// TwinCAT 3 PLC project Linearachse
// ProgramVersion: 3.1.4022.1
// libraries:
//   Tc2_Standard, * (Beckhoff Automation GmbH)
//   Tc2_System, * (Beckhoff Automation GmbH)
//   Tc3_Module, * (Beckhoff Automation GmbH)
// project tree:
//   GVLs/ Sim.TcGVL
//   / PlcTask.TcTTO (not stored)
//   POUs/ Linearachse.TcPOU, MAIN.TcPOU
//   Privat/ DatenRangieren.TcPOU, Hardware.TcGVL, Computer.TcGVL
// real-time tasks:
//   TASK PlcTask: cycle T#10ms, priority 20, ADS port 350
// motion (NC):
//   TASK NC-Task 1 SAF: cycle T#2ms, priority 4, ADS port 501
//   TASK NC-Task 1 SVB: cycle T#10ms, priority 8, ADS port 511
//   AXIS Axis 1 (id 1)
//     OtherSettings: AllowMotionCmdToSlave=true
//     encoder EncType=4
//       EncPara: MaxCount=#x0000ffff
//         Inc: RefSoftSyncMask=#x0000ffff
//     drive DrvType=24
//       Analog: ScaleFactorActTorque=0.1
//       TimeComp: TaskDelayCycles=1
//     controller CtrType=1
//       CtrPara: PriorControlFactor=1
//         Observer: BandWidth=20
//   AXIS Axis 2 (id 2)
//     OtherSettings: AllowMotionCmdToSlave=true
//     encoder EncType=4
//       EncPara: MaxCount=#x0000ffff
//         Inc: RefSoftSyncMask=#x0000ffff
//     drive DrvType=24
//       Analog: ScaleFactorActTorque=0.1
//       TimeComp: TaskDelayCycles=1
//     controller CtrType=1
//       CtrPara: PriorControlFactor=1
//         Observer: BandWidth=20
//   AXIS Axis 3 (id 3)
//     OtherSettings: AllowMotionCmdToSlave=true
//     encoder EncType=4
//       EncPara: MaxCount=#x0000ffff
//     drive DrvType=23
//       Analog: ScaleFactorActTorque=0.1
//       TimeComp: TaskDelayCycles=1
//     controller CtrType=1
//       CtrPara: PriorControlFactor=1
//         Observer: BandWidth=20
//   AXIS Axis 4 (id 4)
//     OtherSettings: AllowMotionCmdToSlave=true
//     encoder EncType=4
//       EncPara: MaxCount=#x0000ffff
//     drive DrvType=23
//       Analog: ScaleFactorActTorque=0.1
//       TimeComp: TaskDelayCycles=1
//     controller CtrType=1
//       CtrPara: PriorControlFactor=1
//         Observer: BandWidth=20
//   AXIS Axis 5 (id 5)
//     OtherSettings: AllowMotionCmdToSlave=true
//     encoder EncType=19
//       EncPara: MaxCount=#xffffffff
//     drive DrvType=16
//       DrvPara: MaxCount=#xffffffff
//         Analog: ScaleFactorActTorque=0.1
//         TimeComp: TaskDelayCycles=1
//     controller CtrType=1
//       CtrPara: PriorControlFactor=1
//         Observer: BandWidth=20
//   AXIS Axis 6 (id 6)
//     OtherSettings: AllowMotionCmdToSlave=true
//     encoder EncType=19
//       EncPara: MaxCount=#xffffffff
//     drive DrvType=16
//       DrvPara: MaxCount=#xffffffff
//         Analog: ScaleFactorActTorque=0.1
//         TimeComp: TaskDelayCycles=1
//     controller CtrType=1
//       CtrPara: PriorControlFactor=1
//         Observer: BandWidth=20
// I/O:
//   DEVICE Device 1 (EtherCAT), AmsNetId 192.168.0.200.2.1
//     Term 1 (EK1200) [EK1200-5000 EtherCAT Power supply (2A E-Bus)]
//       Term 2 (EL1809) [EL1809 16Ch. Dig. Input 24V, 3ms]
//       Term 3 (EL1809) [EL1809 16Ch. Dig. Input 24V, 3ms]
//       Term 4 (EL2809) [EL2809 16Ch. Dig. Output 24V, 0.5A]
//       Term 5 (EL2809) [EL2809 16Ch. Dig. Output 24V, 0.5A]
//       Term 6 (EL3064) [EL3064 4Ch. Ana. Input 0-10V]
//       Term 7 (EL4034) [EL4034 4Ch. Ana. Output +/-10V, 12bit]
//       Term 8 (EL7031) [EL7031 1Ch. Stepper motor output stage (24V, 1.5A)]
//       Term 9 (EL7031) [EL7031 1Ch. Stepper motor output stage (24V, 1.5A)]
//       Term 10 (EL7332) [EL7332 2Ch. DC motor output stage (24V, 1.5A)]
//       Term 11 (EL7201-0010) [EL7201-0010 1Ch. MDP742 Servo motor output stage with OCT (50V, 4A)]
//       Term 12 (EL7201-0010) [EL7201-0010 1Ch. MDP742 Servo motor output stage with OCT (50V, 4A)]
//       Term 26 (EL6090) [EL6090 Display terminal]
//       Term 27 (EK1110) [EK1110 EtherCAT extension]
// variable links:
//   NC-Task 1 SAF/Axes/Axis 1 <-> Device 1 (EtherCAT)/Term 1 (EK1200)/Term 8 (EL7031)
//     Drive/Inputs/In/nState1 @bit 3 <-> STM Status/Status/Error
//     Drive/Inputs/In/nState1 @bit 5 <-> STM Status/Status/Moving negative
//     Drive/Inputs/In/nState1 @bit 4 <-> STM Status/Status/Moving positive
//     Drive/Inputs/In/nState1 @bit 1 <-> STM Status/Status/Ready
//     Drive/Inputs/In/nState1 <-> STM Status/Status/Ready to enable
//     Drive/Inputs/In/nState1 @bit 6 <-> STM Status/Status/Torque reduced
//     Drive/Inputs/In/nState1 @bit 2 <-> STM Status/Status/Warning
//     Drive/Inputs/In/nState2 @bit 3 <-> STM Status/Status/Digital input 1
//     Drive/Inputs/In/nState2 @bit 4 <-> STM Status/Status/Digital input 2
//     Drive/Inputs/In/nState2 @bit 5 <-> STM Status/Status/Sync error
//     Drive/Inputs/In/nState2 @bit 7 <-> STM Status/Status/TxPDO Toggle
//     Drive/Inputs/In/nState4 @bit 1 <-> WcState/InputToggle
//     Drive/Inputs/In/nState4 <-> WcState/WcState
//     Drive/Outputs/Out/nCtrl1 <-> STM Control/Control/Enable
//     Drive/Outputs/Out/nCtrl1 @bit 2 <-> STM Control/Control/Reduce torque
//     Drive/Outputs/Out/nCtrl1 @bit 1 <-> STM Control/Control/Reset
//     Drive/Outputs/Out/nDataOut2[0] <-> STM Velocity/Velocity
//     Enc/Inputs/In/nDataIn1[0] <-> ENC Status compact/Counter value
//     Enc/Inputs/In/nDataIn2[0] <-> ENC Status compact/Latch value
//     Enc/Inputs/In/nState1 @bit 4 <-> ENC Status compact/Status/Counter overflow
//     Enc/Inputs/In/nState1 @bit 3 <-> ENC Status compact/Status/Counter underflow
//     Enc/Inputs/In/nState1 @bit 1 <-> ENC Status compact/Status/Latch extern valid
//     Enc/Inputs/In/nState1 @bit 2 <-> ENC Status compact/Status/Set counter done
//     Enc/Inputs/In/nState2 @bit 4 <-> ENC Status compact/Status/Status of extern latch
//     Enc/Inputs/In/nState2 @bit 5 <-> ENC Status compact/Status/Sync error
//     Enc/Inputs/In/nState2 @bit 7 <-> ENC Status compact/Status/TxPDO Toggle
//     Enc/Inputs/In/nState4 @bit 1 <-> WcState/InputToggle
//     Enc/Inputs/In/nState4 <-> WcState/WcState
//     Enc/Outputs/Out/nCtrl1 @bit 3 <-> ENC Control compact/Control/Enable latch extern on negative edge
//     Enc/Outputs/Out/nCtrl1 @bit 1 <-> ENC Control compact/Control/Enable latch extern on positive edge
//     Enc/Outputs/Out/nCtrl1 @bit 2 <-> ENC Control compact/Control/Set counter
//     Enc/Outputs/Out/nDataOut1[0] <-> ENC Control compact/Set counter value
//   NC-Task 1 SAF/Axes/Axis 2 <-> Device 1 (EtherCAT)/Term 1 (EK1200)/Term 9 (EL7031)
//     Drive/Inputs/In/nState1 @bit 3 <-> STM Status/Status/Error
//     Drive/Inputs/In/nState1 @bit 5 <-> STM Status/Status/Moving negative
//     Drive/Inputs/In/nState1 @bit 4 <-> STM Status/Status/Moving positive
//     Drive/Inputs/In/nState1 @bit 1 <-> STM Status/Status/Ready
//     Drive/Inputs/In/nState1 <-> STM Status/Status/Ready to enable
//     Drive/Inputs/In/nState1 @bit 6 <-> STM Status/Status/Torque reduced
//     Drive/Inputs/In/nState1 @bit 2 <-> STM Status/Status/Warning
//     Drive/Inputs/In/nState2 @bit 3 <-> STM Status/Status/Digital input 1
//     Drive/Inputs/In/nState2 @bit 4 <-> STM Status/Status/Digital input 2
//     Drive/Inputs/In/nState2 @bit 5 <-> STM Status/Status/Sync error
//     Drive/Inputs/In/nState2 @bit 7 <-> STM Status/Status/TxPDO Toggle
//     Drive/Inputs/In/nState4 @bit 1 <-> WcState/InputToggle
//     Drive/Inputs/In/nState4 <-> WcState/WcState
//     Drive/Outputs/Out/nCtrl1 <-> STM Control/Control/Enable
//     Drive/Outputs/Out/nCtrl1 @bit 2 <-> STM Control/Control/Reduce torque
//     Drive/Outputs/Out/nCtrl1 @bit 1 <-> STM Control/Control/Reset
//     Drive/Outputs/Out/nDataOut2[0] <-> STM Velocity/Velocity
//     Enc/Inputs/In/nDataIn1[0] <-> ENC Status compact/Counter value
//     Enc/Inputs/In/nDataIn2[0] <-> ENC Status compact/Latch value
//     Enc/Inputs/In/nState1 @bit 4 <-> ENC Status compact/Status/Counter overflow
//     Enc/Inputs/In/nState1 @bit 3 <-> ENC Status compact/Status/Counter underflow
//     Enc/Inputs/In/nState1 @bit 1 <-> ENC Status compact/Status/Latch extern valid
//     Enc/Inputs/In/nState1 @bit 2 <-> ENC Status compact/Status/Set counter done
//     Enc/Inputs/In/nState2 @bit 4 <-> ENC Status compact/Status/Status of extern latch
//     Enc/Inputs/In/nState2 @bit 5 <-> ENC Status compact/Status/Sync error
//     Enc/Inputs/In/nState2 @bit 7 <-> ENC Status compact/Status/TxPDO Toggle
//     Enc/Inputs/In/nState4 @bit 1 <-> WcState/InputToggle
//     Enc/Inputs/In/nState4 <-> WcState/WcState
//     Enc/Outputs/Out/nCtrl1 @bit 3 <-> ENC Control compact/Control/Enable latch extern on negative edge
//     Enc/Outputs/Out/nCtrl1 @bit 1 <-> ENC Control compact/Control/Enable latch extern on positive edge
//     Enc/Outputs/Out/nCtrl1 @bit 2 <-> ENC Control compact/Control/Set counter
//     Enc/Outputs/Out/nDataOut1[0] <-> ENC Control compact/Set counter value
//   NC-Task 1 SAF/Axes/Axis 3 <-> Device 1 (EtherCAT)/Term 1 (EK1200)/Term 10 (EL7332)
//     Drive/Inputs/In/nState1 @bit 3 <-> DCM Status Channel 1/Status/Error
//     Drive/Inputs/In/nState1 @bit 5 <-> DCM Status Channel 1/Status/Moving negative
//     Drive/Inputs/In/nState1 @bit 4 <-> DCM Status Channel 1/Status/Moving positive
//     Drive/Inputs/In/nState1 @bit 1 <-> DCM Status Channel 1/Status/Ready
//     Drive/Inputs/In/nState1 <-> DCM Status Channel 1/Status/Ready to enable
//     Drive/Inputs/In/nState1 @bit 6 <-> DCM Status Channel 1/Status/Torque reduced
//     Drive/Inputs/In/nState1 @bit 2 <-> DCM Status Channel 1/Status/Warning
//     Drive/Inputs/In/nState2 @bit 3 <-> DCM Status Channel 1/Status/Digital input 1
//     Drive/Inputs/In/nState2 @bit 4 <-> DCM Status Channel 1/Status/Digital input 2
//     Drive/Inputs/In/nState2 @bit 5 <-> DCM Status Channel 1/Status/Sync error
//     Drive/Inputs/In/nState2 @bit 7 <-> DCM Status Channel 1/Status/TxPDO Toggle
//     Drive/Inputs/In/nState4 @bit 1 <-> WcState/InputToggle
//     Drive/Inputs/In/nState4 <-> WcState/WcState
//     Drive/Outputs/Out/nCtrl1 <-> DCM Control Channel 1/Control/Enable
//     Drive/Outputs/Out/nCtrl1 @bit 2 <-> DCM Control Channel 1/Control/Reduce torque
//     Drive/Outputs/Out/nCtrl1 @bit 1 <-> DCM Control Channel 1/Control/Reset
//     Drive/Outputs/Out/nDataOut2[0] <-> DCM Velocity Channel 1/Velocity
//   NC-Task 1 SAF/Axes/Axis 4 <-> Device 1 (EtherCAT)/Term 1 (EK1200)/Term 10 (EL7332)
//     Drive/Inputs/In/nState1 @bit 3 <-> DCM Status Channel 2/Status/Error
//     Drive/Inputs/In/nState1 @bit 5 <-> DCM Status Channel 2/Status/Moving negative
//     Drive/Inputs/In/nState1 @bit 4 <-> DCM Status Channel 2/Status/Moving positive
//     Drive/Inputs/In/nState1 @bit 1 <-> DCM Status Channel 2/Status/Ready
//     Drive/Inputs/In/nState1 <-> DCM Status Channel 2/Status/Ready to enable
//     Drive/Inputs/In/nState1 @bit 6 <-> DCM Status Channel 2/Status/Torque reduced
//     Drive/Inputs/In/nState1 @bit 2 <-> DCM Status Channel 2/Status/Warning
//     Drive/Inputs/In/nState2 @bit 3 <-> DCM Status Channel 2/Status/Digital input 1
//     Drive/Inputs/In/nState2 @bit 4 <-> DCM Status Channel 2/Status/Digital input 2
//     Drive/Inputs/In/nState2 @bit 5 <-> DCM Status Channel 2/Status/Sync error
//     Drive/Inputs/In/nState2 @bit 7 <-> DCM Status Channel 2/Status/TxPDO Toggle
//     Drive/Inputs/In/nState4 @bit 1 <-> WcState/InputToggle
//     Drive/Inputs/In/nState4 <-> WcState/WcState
//     Drive/Outputs/Out/nCtrl1 <-> DCM Control Channel 2/Control/Enable
//     Drive/Outputs/Out/nCtrl1 @bit 2 <-> DCM Control Channel 2/Control/Reduce torque
//     Drive/Outputs/Out/nCtrl1 @bit 1 <-> DCM Control Channel 2/Control/Reset
//     Drive/Outputs/Out/nDataOut2[0] <-> DCM Velocity Channel 2/Velocity
//   NC-Task 1 SAF/Axes/Axis 5 <-> Device 1 (EtherCAT)/Term 1 (EK1200)/Term 11 (EL7201-0010)
//     Drive/Inputs/In/nDcOutputTime <-> InfoData/DcOutputShift
//     Drive/Inputs/In/nState1 <-> DRV Statusword/Statusword
//     Drive/Inputs/In/nState2 <-> DRV Statusword/Statusword @bit 8
//     Drive/Inputs/In/nState4 @bit 1 <-> WcState/InputToggle
//     Drive/Inputs/In/nState4 <-> WcState/WcState
//     Drive/Outputs/Out/nCtrl1 <-> DRV Controlword/Controlword
//     Drive/Outputs/Out/nCtrl2 <-> DRV Controlword/Controlword @bit 8
//     Drive/Outputs/Out/nDataOut2 <-> DRV Target velocity/Target velocity
//     Enc/Inputs/In/nDataIn1 <-> FB Position/Position
//     Enc/Inputs/In/nDcInputTime <-> InfoData/DcInputShift
//     Enc/Inputs/In/nState4 @bit 1 <-> WcState/InputToggle
//     Enc/Inputs/In/nState4 <-> WcState/WcState
//   NC-Task 1 SAF/Axes/Axis 6 <-> Device 1 (EtherCAT)/Term 1 (EK1200)/Term 12 (EL7201-0010)
//     Drive/Inputs/In/nDcOutputTime <-> InfoData/DcOutputShift
//     Drive/Inputs/In/nState1 <-> DRV Statusword/Statusword
//     Drive/Inputs/In/nState2 <-> DRV Statusword/Statusword @bit 8
//     Drive/Inputs/In/nState4 @bit 1 <-> WcState/InputToggle
//     Drive/Inputs/In/nState4 <-> WcState/WcState
//     Drive/Outputs/Out/nCtrl1 <-> DRV Controlword/Controlword
//     Drive/Outputs/Out/nCtrl2 <-> DRV Controlword/Controlword @bit 8
//     Drive/Outputs/Out/nDataOut2 <-> DRV Target velocity/Target velocity
//     Enc/Inputs/In/nDataIn1 <-> FB Position/Position
//     Enc/Inputs/In/nDcInputTime <-> InfoData/DcInputShift
//     Enc/Inputs/In/nState4 @bit 1 <-> WcState/InputToggle
//     Enc/Inputs/In/nState4 <-> WcState/WcState
//   Linearachse/Linearachse Instance <-> Device 1 (EtherCAT)/Term 1 (EK1200)/Term 2 (EL1809)
//     PlcTask Inputs/Hardware.DI_0_1_bis_8 <-> Channel 1/Input
//     PlcTask Inputs/Hardware.DI_0_9_bis_16 <-> Channel 8/Input
//     PlcTask Inputs/Hardware.DI_0_1_bis_8 @bit 1 <-> Channel 2/Input
//     PlcTask Inputs/Hardware.DI_0_1_bis_8 @bit 2 <-> Channel 3/Input
//     PlcTask Inputs/Hardware.DI_0_1_bis_8 @bit 3 <-> Channel 4/Input
//     PlcTask Inputs/Hardware.DI_0_1_bis_8 @bit 4 <-> Channel 5/Input
//     PlcTask Inputs/Hardware.DI_0_1_bis_8 @bit 5 <-> Channel 6/Input
//     PlcTask Inputs/Hardware.DI_0_1_bis_8 @bit 6 <-> Channel 7/Input
//     PlcTask Inputs/Hardware.DI_0_9_bis_16 @bit 1 <-> Channel 10/Input
//     PlcTask Inputs/Hardware.DI_0_9_bis_16 @bit 2 <-> Channel 11/Input
//     PlcTask Inputs/Hardware.DI_0_9_bis_16 @bit 3 <-> Channel 12/Input
//     PlcTask Inputs/Hardware.DI_0_9_bis_16 @bit 4 <-> Channel 13/Input
//     PlcTask Inputs/Hardware.DI_0_9_bis_16 @bit 5 <-> Channel 14/Input
//     PlcTask Inputs/Hardware.DI_0_9_bis_16 @bit 6 <-> Channel 15/Input
//     PlcTask Inputs/Hardware.DI_0_9_bis_16 @bit 7 <-> Channel 16/Input
//   Linearachse/Linearachse Instance <-> Device 1 (EtherCAT)/Term 1 (EK1200)/Term 3 (EL1809)
//     PlcTask Inputs/Hardware.DI_1_1_bis_8 <-> Channel 1/Input
//     PlcTask Inputs/Hardware.DI_1_9_bis_16 <-> Channel 9/Input
//     PlcTask Inputs/Hardware.DI_1_1_bis_8 @bit 1 <-> Channel 2/Input
//     PlcTask Inputs/Hardware.DI_1_1_bis_8 @bit 2 <-> Channel 3/Input
//     PlcTask Inputs/Hardware.DI_1_1_bis_8 @bit 3 <-> Channel 4/Input
//     PlcTask Inputs/Hardware.DI_1_1_bis_8 @bit 4 <-> Channel 5/Input
//     PlcTask Inputs/Hardware.DI_1_1_bis_8 @bit 5 <-> Channel 6/Input
//     PlcTask Inputs/Hardware.DI_1_1_bis_8 @bit 6 <-> Channel 7/Input
//     PlcTask Inputs/Hardware.DI_1_1_bis_8 @bit 7 <-> Channel 8/Input
//     PlcTask Inputs/Hardware.DI_1_9_bis_16 @bit 1 <-> Channel 10/Input
//     PlcTask Inputs/Hardware.DI_1_9_bis_16 @bit 2 <-> Channel 11/Input
//     PlcTask Inputs/Hardware.DI_1_9_bis_16 @bit 3 <-> Channel 12/Input
//     PlcTask Inputs/Hardware.DI_1_9_bis_16 @bit 4 <-> Channel 13/Input
//     PlcTask Inputs/Hardware.DI_1_9_bis_16 @bit 5 <-> Channel 14/Input
//     PlcTask Inputs/Hardware.DI_1_9_bis_16 @bit 6 <-> Channel 15/Input
//     PlcTask Inputs/Hardware.DI_1_9_bis_16 @bit 7 <-> Channel 16/Input
//   Linearachse/Linearachse Instance <-> Device 1 (EtherCAT)/Term 1 (EK1200)/Term 4 (EL2809)
//     PlcTask Outputs/Hardware.DQ_0_1_bis_8 <-> Channel 1/Output
//     PlcTask Outputs/Hardware.DQ_0_9_bis_16 <-> Channel 9/Output
//     PlcTask Outputs/Hardware.DQ_0_1_bis_8 @bit 1 <-> Channel 2/Output
//     PlcTask Outputs/Hardware.DQ_0_1_bis_8 @bit 2 <-> Channel 3/Output
//     PlcTask Outputs/Hardware.DQ_0_1_bis_8 @bit 3 <-> Channel 4/Output
//     PlcTask Outputs/Hardware.DQ_0_1_bis_8 @bit 4 <-> Channel 5/Output
//     PlcTask Outputs/Hardware.DQ_0_1_bis_8 @bit 5 <-> Channel 6/Output
//     PlcTask Outputs/Hardware.DQ_0_1_bis_8 @bit 6 <-> Channel 7/Output
//     PlcTask Outputs/Hardware.DQ_0_1_bis_8 @bit 7 <-> Channel 8/Output
//     PlcTask Outputs/Hardware.DQ_0_9_bis_16 @bit 1 <-> Channel 10/Output
//     PlcTask Outputs/Hardware.DQ_0_9_bis_16 @bit 2 <-> Channel 11/Output
//     PlcTask Outputs/Hardware.DQ_0_9_bis_16 @bit 3 <-> Channel 12/Output
//     PlcTask Outputs/Hardware.DQ_0_9_bis_16 @bit 4 <-> Channel 13/Output
//     PlcTask Outputs/Hardware.DQ_0_9_bis_16 @bit 5 <-> Channel 14/Output
//     PlcTask Outputs/Hardware.DQ_0_9_bis_16 @bit 6 <-> Channel 15/Output
//     PlcTask Outputs/Hardware.DQ_0_9_bis_16 @bit 7 <-> Channel 16/Output
//   Linearachse/Linearachse Instance <-> Device 1 (EtherCAT)/Term 1 (EK1200)/Term 5 (EL2809)
//     PlcTask Outputs/Hardware.DQ_1_1_bis_8 <-> Channel 1/Output
//     PlcTask Outputs/Hardware.DQ_1_9_bis_16 <-> Channel 9/Output
//     PlcTask Outputs/Hardware.DQ_1_1_bis_8 @bit 1 <-> Channel 2/Output
//     PlcTask Outputs/Hardware.DQ_1_1_bis_8 @bit 2 <-> Channel 3/Output
//     PlcTask Outputs/Hardware.DQ_1_1_bis_8 @bit 3 <-> Channel 4/Output
//     PlcTask Outputs/Hardware.DQ_1_1_bis_8 @bit 4 <-> Channel 5/Output
//     PlcTask Outputs/Hardware.DQ_1_1_bis_8 @bit 5 <-> Channel 6/Output
//     PlcTask Outputs/Hardware.DQ_1_1_bis_8 @bit 6 <-> Channel 7/Output
//     PlcTask Outputs/Hardware.DQ_1_1_bis_8 @bit 7 <-> Channel 8/Output
//     PlcTask Outputs/Hardware.DQ_1_9_bis_16 @bit 1 <-> Channel 10/Output
//     PlcTask Outputs/Hardware.DQ_1_9_bis_16 @bit 2 <-> Channel 11/Output
//     PlcTask Outputs/Hardware.DQ_1_9_bis_16 @bit 3 <-> Channel 12/Output
//     PlcTask Outputs/Hardware.DQ_1_9_bis_16 @bit 4 <-> Channel 13/Output
//     PlcTask Outputs/Hardware.DQ_1_9_bis_16 @bit 5 <-> Channel 14/Output
//     PlcTask Outputs/Hardware.DQ_1_9_bis_16 @bit 6 <-> Channel 15/Output
//     PlcTask Outputs/Hardware.DQ_1_9_bis_16 @bit 7 <-> Channel 16/Output
//   Linearachse/Linearachse Instance <-> Device 1 (EtherCAT)/Term 1 (EK1200)/Term 6 (EL3064)
//     PlcTask Inputs/Hardware.AI_0_{1..4} <-> AI Standard Channel {1..4}/Value  (4 links)
//   Linearachse/Linearachse Instance <-> Device 1 (EtherCAT)/Term 1 (EK1200)/Term 7 (EL4034)
//     PlcTask Outputs/Hardware.AQ_0_{1..4} <-> AO Outputs Channel {1..4}/Analog output  (4 links)

// ---- GVLs/Sim.TcGVL
{attribute 'qualified_only'}
VAR_GLOBAL
	
	// Linearantrieb Endlage links (Öffner)
	B1 AT %I*: BOOL; 
	// Linearantrieb Endlage rechts (Öffner)
	B2 AT %I*: BOOL;
	// Taster (1) (Schliesser)
	S1 AT %I*: BOOL;	
	// Taster (0) (Öffner)
	S2 AT %I*: BOOL;
	// Taster I (Schliesser)
	S3 AT %I*: BOOL;
	// Taster II (Schliesser)
	S4 AT %I*: BOOL;
	// Taster Pfeil auf (Schliesser)
	S5 AT %I*: BOOL;
	// Taster Pfeil ab (Schliesser)
	S6 AT %I*: BOOL;
	// Taster + (Schliesser)
	S7 AT %I*: BOOL;
	// Taster - (Schliesser)
	S8 AT %I*: BOOL;
	// Taster STOP (Öffner)
	S9 AT %I*: BOOL;
	// Taster Not Halt (Öffner)
	S10 AT %I*: BOOL;
	// Taster Not Halt (Schliesser)
	S11 AT %I*: BOOL;

	// Linearantrieb Rechtslauf
	Q1 AT %Q*: BOOL;
	// Linearantrieb Linkslauf
	Q2 AT %Q*: BOOL;
	// Meldeleuchte im Taster S1 (weiß)
	P1 AT %Q*: BOOL;
	// Meldeleuchte weiß
	P2 AT %Q*: BOOL;
	// Meldeleuchte rot
	P3 AT %Q*: BOOL;
	// Meldeleuchte grün
	P4 AT %Q*: BOOL;

END_VAR

// ---- Privat/Hardware.TcGVL
{attribute 'qualified_only'}
VAR_GLOBAL
	// Digitale Eingänge EL1809
	DI_0_1_bis_8 AT %I*: BYTE; 	//dSub 25 Stecker	Term 2
	DI_0_9_bis_16 AT %I*: BYTE; //dSub 25 Stecker	Term 2
	DI_1_1_bis_8 AT %I*: BYTE; 	//					Term 3
	DI_1_9_bis_16 AT %I*: BYTE; //					Term 3
	
	// Digitale Ausgänge EL2809
	DQ_0_1_bis_8 AT %Q*: BYTE; 	//dSub 25 Stecker	Term 4
	DQ_0_9_bis_16 AT %Q*: BYTE; //dSub 25 Stecker	Term 4
	DQ_1_1_bis_8 AT %Q*: BYTE; 	//					Term 5
	DQ_1_9_bis_16 AT %Q*: BYTE; //					Term 5
	
	// Analoge Eingänge EL3064
	AI_0_1 AT %I*: INT;			//					Term 6
	AI_0_2 AT %I*: INT;			//					Term 6
	AI_0_3 AT %I*: INT;			//					Term 6
	AI_0_4 AT %I*: INT;			//					Term 6
	
	// Analoge Ausgänge EL4034
	AQ_0_1 AT %Q*: INT;			//					Term 7
	AQ_0_2 AT %Q*: INT;			//					Term 7
	AQ_0_3 AT %Q*: INT;			//					Term 7
	AQ_0_4 AT %Q*: INT;			//					Term 7
	
END_VAR

// ---- Privat/Computer.TcGVL
{attribute 'qualified_only'}
VAR_GLOBAL
	AnInput : ARRAY[0..100] OF INT;
	AnOutput : ARRAY[0..100] OF INT;
	DigInput : ARRAY[0..100] OF BYTE;	
	DigOutput : ARRAY[0..100] OF BYTE;
	SimulationAktiv:BOOL;
	Versionsbezeichnung: STRING := 'Labor Linearachse V2.0';
END_VAR

// ---- POUs/Linearachse.TcPOU
FUNCTION_BLOCK Linearachse
VAR_INPUT
END_VAR
VAR_OUTPUT
END_VAR
VAR
END_VAR

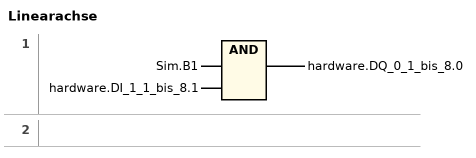
// NETWORK 1
hardware.DQ_0_1_bis_8.0 := Sim.B1 AND hardware.DI_1_1_bis_8.1;

// NETWORK 2

END_FUNCTION_BLOCK

// ---- POUs/MAIN.TcPOU
PROGRAM MAIN
VAR
	LinearAchse: Linearachse;
END_VAR

DatenRangieren();
LinearAchse();

END_PROGRAM

// ---- Privat/DatenRangieren.TcPOU
FUNCTION DatenRangieren : BOOL
VAR_INPUT
END_VAR
VAR
END_VAR

IF (Computer.SimulationAktiv = TRUE) THEN
;	// es werden die Daten von den Arrays verwendet
ELSE
	Computer.DigInput[0] := Hardware.DI_0_1_bis_8;
	Computer.DigInput[1] := Hardware.DI_0_9_bis_16;
	Computer.DigInput[2] := Hardware.DI_1_1_bis_8;
	Computer.DigInput[3] := Hardware.DI_1_9_bis_16;
	
	Hardware.DQ_0_1_bis_8 := Computer.DigInput[0];
	Hardware.DQ_0_9_bis_16 := Computer.DigInput[1];
	Hardware.DQ_1_1_bis_8 := Computer.DigInput[2];
	Hardware.DQ_1_9_bis_16 := Computer.DigInput[3];
	
	
	Computer.AnInput[0] :=  Hardware.AI_0_1;
	Computer.AnInput[1] :=  Hardware.AI_0_2;
	Computer.AnInput[2] :=  Hardware.AI_0_3;
	Computer.AnInput[3] :=  Hardware.AI_0_4;
	
	Hardware.AQ_0_1 := Computer.AnOutput[0];
	Hardware.AQ_0_2 := Computer.AnOutput[1];
	Hardware.AQ_0_3 := Computer.AnOutput[2];
	Hardware.AQ_0_4 := Computer.AnOutput[3];	
END_IF

Sim.B1:=Computer.DigInput[0].0;

END_FUNCTION
